PROGRAM A21
VAR_IN_OUT
	sectionCIP : ChipboardEx;
	sectionWB : WoodBunkEx;
	
	bundlesQueue : ARRAY[0..Consts.maxQueue] OF Bundle;
	bundlesBypass : ARRAY[0..Consts.maxQueue] OF BOOL;
END_VAR
VAR_OUTPUT //conveyors only
	A21_SC_C18 		: ConveyorSC;
	A21_LSC_C19 	: ConveyorLSC;
	A21_LSC_C20 	: ConveyorLSC;
	A21_LSC_C21 	: ConveyorLSC;
END_VAR
VAR //hardware
	robot1, robot2 : RobotA21;
	toolStorageA21Left, toolStorageA21Right : A21ToolStorage;
	
	skidA21Left, skidA21Right : SkidMagazine;
	magazineA21Left, magazineA21Right : SkidMagazine;
	stagingTableLeft, stagingTableRight : StagingTable;
	strapperA21 : StrapMachine;
	
	horizontalDriveA21Left, horizontalDriveA21Right : AirPiston := (
		limitSensorDefaultState := FALSE,
		useBrake := FALSE);
	
	verticalDriveA21Left, verticalDriveA21Right : ClearLinkMC := (
		limitSensorDefaultState := TRUE, 
		homingDirectionOut := TRUE, //outwards (up)
		minPosition := 0,
		displacementPerRotation := 1,
		unitsPerPulse := 8000); //0.1x gearbox, 10 revs/pulse to compensate
		
	insertionA21Left, insertionA21Right : Insertion;
	
	pistonA21Bottom : SimplePiston;
	
	suctionA21Top : ARRAY[1..3] OF SuctionPad;
	suctionA21Left : ARRAY[1..4] OF SuctionPad;
	suctionA21Right : ARRAY[1..4] OF SuctionPad; 
	suctionA21Bottom : ARRAY[1..2] OF SuctionPad;
END_VAR
VAR //material holder arrays
	skidSlotsA21Left, skidSlotsA21Right AT %M* : ARRAY[1..2] OF MaterialSlot;
	magazineSlotsA21Left, magazineSlotsA21Right AT %M* : ARRAY[1..15] OF MaterialSlot;
	tableSlotsA21Left, tableSlotsA21Right : ARRAY[1..10] OF MaterialSlot;
	(*
	different material holders have different capacities
	arrays are declared here and passed into material holder instances by reference
	direct access to these arrays is strongly discouraged
	
	arrays of slots are used to display the data on TcHmi datagrids in slot-occupancy struct format
	*)
END_VAR
VAR //statuses and alarms
	stackLightCIP : PMLStackLight; //chipboard stack light
	stackLightWB : PMLStackLight; //wood bunk stack light
	
	panelPowerOn : BOOL;
	safetyOk : BOOL;
	airPressureOk : BOOL;
END_VAR
VAR //other
	conveyorsCIP : ARRAY[1..3] OF POINTER TO ConveyorSC;
	conveyorsWB : ARRAY[1..1] OF POINTER TO ConveyorSC;
END_VAR

callHardware();

setupHardware();

runModules();

callHardware();

METHOD PRIVATE callHardware : BOOL
{warning disable C0371}

robot1(strapSafety := (NOT strapperA21.enable AND NOT strapperA21.execute AND strapperA21.home));	
robot2(strapSafety := (NOT strapperA21.enable AND NOT strapperA21.execute AND strapperA21.home));

skidA21Left(slots := skidSlotsA21Left);
skidA21Right(slots := skidSlotsA21Right);

stagingTableLeft(slots := tableSlotsA21Left);
stagingTableRight(slots := tableSlotsA21Right);

magazineA21Left(slots := magazineSlotsA21Left);
magazineA21Right(slots := magazineSlotsA21Right);

strapperA21(extSafety := robot1.strapSafetyIn AND robot2.strapSafetyIn);

verticalDriveA21Left(bEnable := TRUE);
verticalDriveA21Right(bEnable := TRUE);
horizontalDriveA21Left(bEnable := TRUE);
horizontalDriveA21Right(bEnable := TRUE);

insertionA21Left(
	slider:= verticalDriveA21Left, 
	screw:= horizontalDriveA21Left, 
	contact=> , 
	active=> , 
	error=> , 
	home=> , 
	homingComplete=> , 
	sliderPos=> );
	
insertionA21Right(
	slider:= verticalDriveA21Right, 
	screw:= horizontalDriveA21Right, 
	contact=> , 
	active=> , 
	error=> , 
	home=> , 
	homingComplete=> , 
	sliderPos=> );

pistonA21Bottom();

stackLightCIP(
	pmlState:= sectionCIP.pmlState, 
	lowMaterial:= , 
	materialExhausted:= , 
	red=> , 
	yellow=> , 
	blue=> , 
	green=> );
	
stackLightWB(
	pmlState:= sectionWB.pmlState, 
	lowMaterial:= , 
	materialExhausted:= , 
	red=> , 
	yellow=> , 
	blue=> , 
	green=> );

(*
tempLeft := TO_INT(BoolPtrArrayToInteger(arr := stagingTableLeft.occupied, lowerBound := 1, upperBound := 10));
tempLeft.15 := NOT strapperA21.bEnable AND NOT strapperA21.execute;
robot1.setGroup(group := 8, value := tempLeft);

tempRight := TO_INT(BoolPtrArrayToInteger(arr := stagingTableRight.occupied, lowerBound := 1, upperBound := 10));
tempRight.15 := NOT strapperA21.bEnable AND NOT strapperA21.execute;
robot2.setGroup(group := 8, value := tempRight);

*)
END_METHOD

METHOD PRIVATE runModules : BOOL
VAR_INPUT
END_VAR
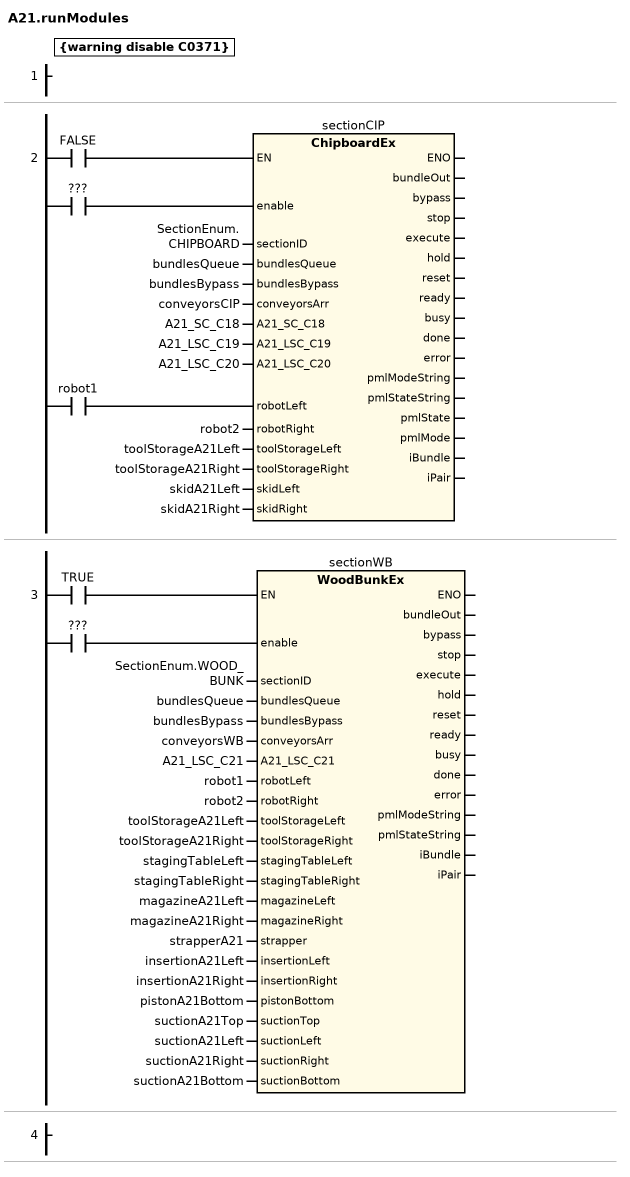
// NETWORK 1
// label: {warning disable C0371}

// NETWORK 2
IF FALSE THEN
    sectionCIP(
        sectionID := SectionEnum.CHIPBOARD,
        bundlesQueue := bundlesQueue,
        bundlesBypass := bundlesBypass,
        conveyorsArr := conveyorsCIP,
        A21_SC_C18 := A21_SC_C18,
        A21_LSC_C19 := A21_LSC_C19,
        A21_LSC_C20 := A21_LSC_C20,
        robotLeft := robot1,
        robotRight := robot2,
        toolStorageLeft := toolStorageA21Left,
        toolStorageRight := toolStorageA21Right,
        skidLeft := skidA21Left,
        skidRight := skidA21Right); // ChipboardEx
END_IF

// NETWORK 3
sectionWB(
    sectionID := SectionEnum.WOOD_BUNK,
    bundlesQueue := bundlesQueue,
    bundlesBypass := bundlesBypass,
    conveyorsArr := conveyorsWB,
    A21_LSC_C21 := A21_LSC_C21,
    robotLeft := robot1,
    robotRight := robot2,
    toolStorageLeft := toolStorageA21Left,
    toolStorageRight := toolStorageA21Right,
    stagingTableLeft := stagingTableLeft,
    stagingTableRight := stagingTableRight,
    magazineLeft := magazineA21Left,
    magazineRight := magazineA21Right,
    strapper := strapperA21,
    insertionLeft := insertionA21Left,
    insertionRight := insertionA21Right,
    pistonBottom := pistonA21Bottom,
    suctionTop := suctionA21Top,
    suctionLeft := suctionA21Left,
    suctionRight := suctionA21Right,
    suctionBottom := suctionA21Bottom); // WoodBunkEx

// NETWORK 4
END_METHOD

METHOD PRIVATE setupHardware : BOOL
VAR
	iWoodBunkSlot : WoodBunk;
	iChipboardSlot : Chipboard;
	i : INT;
END_VAR
FOR iWoodBunkSlot:=1 TO WoodBunk.size-1 BY 1 DO //init wood bunk magazine slots
	magazineA21Left.setSlot(i := iWoodBunkSlot, material := TO_STRING(iWoodBunkSlot), error => );
	magazineA21Right.setSlot(i := iWoodBunkSlot, material := TO_STRING(iWoodBunkSlot), error => );
END_FOR

//--------------------------------------------------

FOR iChipboardSlot:=1 TO Chipboard.size-1 BY 1 DO //init chipboard skid slots
	skidA21Left.setSlot(i := iChipboardSlot, material := TO_STRING(iChipboardSlot), error => );
	skidA21Right.setSlot(i := iChipboardSlot, material := TO_STRING(iChipboardSlot), error => );
END_FOR

//--------------------------------------------------

FOR i:=1 TO Consts.maxQueue BY 1 DO //get wood bunk magazine + chipboard skid availability from robot1 and robot2
	{warning disable C0195}
	skidA21Left.setOccupancy( i := i, occupancy := IntegerBitAccess(robot1.inputs[4], i-1) );
	skidA21Right.setOccupancy( i := i, occupancy := IntegerBitAccess(robot2.inputs[4], i-1) );

	magazineA21Left.setOccupancy( i := i, occupancy := IntegerBitAccess(robot1.inputs[3], i-1) );
	magazineA21Right.setOccupancy( i := i, occupancy := IntegerBitAccess(robot2.inputs[3], i-1) );
END_FOR

//--------------------------------------------------
conveyorsCIP[1] := ADR(A21_SC_C18);
conveyorsCIP[2] := ADR(A21_LSC_C19);
conveyorsCIP[3] := ADR(A21_LSC_C20);

conveyorsWB[1] := ADR(A21_LSC_C21);
END_METHOD

END_PROGRAM

(* stored: Version 1.1.0.1, ProductVersion 3.1.4024.11
   POU A21: Id {21b63919-ed47-4b37-9367-110a5a725bc2}, SpecialFunc None
   Method callHardware: Id {cbd6668a-4a61-4a31-9125-2161ec10dadd}
   Method runModules: Id {a7d94c7f-07fb-4636-88b8-1660b818a96f}
   Method setupHardware: Id {07421a38-8a2e-44b7-8418-15ab376e1b51} *)
